INTERFACE I_AmeClient

METHOD OnNewMsgToSend
END_METHOD

METHOD OnNewRcvMsg
END_METHOD

END_INTERFACE

(* stored: Version 1.1.0.1
   Itf I_AmeClient: Id {331a3e02-f3d3-4b18-a5d7-9910e6c08ce3}
   Folder Events: Id {4bfd18d6-0d8b-46e7-abb3-bee0ee031d13}
   Method OnNewMsgToSend: Id {c7816cc3-c669-4d59-9b66-c8de47aaa824}
   Method OnNewRcvMsg: Id {e644f43b-bb71-4cff-943b-b1f9cc8459fa} *)
